Staubli VAL3: moveBox.pjx

--- moveBox.pjx ---
Parameters version=s7.11.2 stackSize=5000 millimeterUnit=true
Program file=start.pgx
Program file=stop.pgx
Data file=moveBox.dtx

--- start.pgx ---
program start()
begin

end
